{attribute 'linkalways'} 
{attribute 'no_explicit_call' := 'This FB is a CLASS and must be accessed using methods or properties'}
{attribute 'enable_dynamic_creation'}
FUNCTION_BLOCK _ETcVnSvmKernelType EXTENDS EnumDatatypeBase
VAR
	localData : ETcVnSvmKernelType;
	activeData : REFERENCE TO ETcVnSvmKernelType;
	enumBaseDatatype : _DINT(localData);
END_VAR

METHOD PRIVATE AddLocalEnumeration
VAR_INPUT
	Enumeration : T_MAXSTRING;
	Value : ETcVnSvmKernelType;
END_VAR
AddEnumeration(Enumeration, Value);
END_METHOD

PROPERTY PUBLIC Address : PVOID
GET
Address := ADR(activeData);
END_GET
END_PROPERTY

METHOD PUBLIC ClearReference
VAR_INPUT
END_VAR
activeData REF= localData;
SetBaseDatatypeReference();
END_METHOD

METHOD PUBLIC Clone : I_Datatype
VAR
    pClone : POINTER TO _ETcVnSvmKernelType;
END_VAR
pClone := __NEW(_ETcVnSvmKernelType(InitialValue := Value));
Clone := pClone^;
END_METHOD

METHOD FB_init : BOOL
VAR_INPUT
	bInitRetains : BOOL; // if TRUE, the retain variables are initialized (warm start / cold start)
	bInCopyCode : BOOL;  // if TRUE, the instance afterwards gets moved into the copy code (online change)
	InitialValue : ETcVnSvmKernelType;
END_VAR
localData := InitialValue;
AddBaseDatatype(enumBaseDatatype);
ClearReference();

AddLocalEnumeration('TCVN_SKT_LINEAR', ETcVnSvmKernelType.TCVN_SKT_LINEAR);
AddLocalEnumeration('TCVN_SKT_POLY', ETcVnSvmKernelType.TCVN_SKT_POLY);
AddLocalEnumeration('TCVN_SKT_RBF', ETcVnSvmKernelType.TCVN_SKT_RBF);
AddLocalEnumeration('TCVN_SKT_SIGMOID', ETcVnSvmKernelType.TCVN_SKT_SIGMOID);
AddLocalEnumeration('TCVN_SKT_CHI2', ETcVnSvmKernelType.TCVN_SKT_CHI2);
AddLocalEnumeration('TCVN_SKT_INTER', ETcVnSvmKernelType.TCVN_SKT_INTER);
END_METHOD

PROPERTY PUBLIC Identifier : T_MAXSTRING
GET
Identifier := 'ETcVnSvmKernelType';
END_GET
END_PROPERTY

METHOD IsEnumeratorValueEqual : BOOL
VAR_INPUT
	Enumerator : I_KeyValueForwardEnumerator;
END_VAR
VAR
	storedValue : ETcVnSvmKernelType;
END_VAR
IF NOT Enumerator.TryGet(storedValue) THEN
	RETURN;
END_IF

IsEnumeratorValueEqual := storedValue = activeData;
END_METHOD

METHOD PUBLIC MakeReferenceTo
VAR_INPUT
	ReferenceTarget : REFERENCE TO ETcVnSvmKernelType;
END_VAR
activeData REF= ReferenceTarget;
SetBaseDatatypeReference();
END_METHOD

METHOD PROTECTED SetBaseDatatypeReference
VAR_INPUT
END_VAR
enumBaseDatatype.MakeReferenceTo(activeData);
END_METHOD

PROPERTY PUBLIC Size : UDINT
GET
Size := SIZEOF(activeData);
END_GET
END_PROPERTY

METHOD TryMakeReferenceTo : BOOL
VAR_INPUT
	Target : I_Datatype;
END_VAR
VAR
	targetAsEnum : I_EnumDatatype;
	pTargetData : POINTER TO ETcVnSvmKernelType;
END_VAR
IF NOT Target.TryResolveAsEnumDatatype(targetAsEnum) THEN
	RETURN;
END_IF

IF targetAsEnum.Identifier <> Identifier THEN
	RETURN;
END_IF

pTargetData := Target.Address;
activeData REF= pTargetData^;
SetBaseDatatypeReference();
TryMakeReferenceTo := TRUE;
END_METHOD

PROPERTY PUBLIC Value : ETcVnSvmKernelType
GET
Value := activeData;
END_GET
SET
activeData := Value;
END_SET
END_PROPERTY

END_FUNCTION_BLOCK

(* stored: Version 1.1.0.1, ProductVersion 3.1.4024.13
   POU _ETcVnSvmKernelType: Id {d4918786-9cab-0cd6-2fcd-e628cd260273}, SpecialFunc None
   Folder Core: Id {512a4051-ce2d-08e0-3e05-45e6bff0025f}
   Folder Protected: Id {379efe20-a124-08ea-22a7-6ae65a05b89e}
   Folder Customize: Id {7ddb8890-7a2c-0ed9-32eb-8c3c1c2fa97c}
   Folder Constructor: Id {fcd5a4ca-c91d-0612-381f-e7e0e9d08047}
   Folder Private: Id {a9a80b6c-e641-03d0-2fa3-3e3ca7077f62}
   Folder Protected: Id {14f43d9a-4447-0614-0f11-bc60955d242b}
   Method AddLocalEnumeration: Id {b036fb34-c348-0c26-0e4c-9bda6ad7c67e}
   Property Address: Id {3cfcd777-4d74-0e79-1921-bcf5dc950f09}
   Get Get: Id {e96f154e-1a78-05de-23c4-a4aac86c2fc4}
   Method ClearReference: Id {2076ad69-a159-003c-045c-402f3267fda5}
   Method Clone: Id {62c5445e-85ae-0278-1045-f8b20dd75b01}
   Method FB_init: Id {363200be-d448-0413-224b-f9a2fa2c8541}
   Property Identifier: Id {7c1918a0-1ef6-05d7-146a-7ab05e9d0811}
   Get Get: Id {8d07742d-cd78-0be9-13ee-6c2f10d61f0c}
   Method IsEnumeratorValueEqual: Id {3e0367b2-34ba-06b7-3e5e-291ef48b21d8}
   Method MakeReferenceTo: Id {b1896ce3-d302-0310-2aec-ad9469df1070}
   Method SetBaseDatatypeReference: Id {e7b57660-8a96-0b5c-32c7-d6f0f74f2b6b}
   Property Size: Id {b05405a8-55d0-028f-3ba3-3c3d630b435e}
   Get Get: Id {759c2f2d-e774-0ab8-2a71-4d3239b7c561}
   Method TryMakeReferenceTo: Id {5537f957-8a00-05e1-2fa4-f921464ca333}
   Property Value: Id {9d332358-2bbb-0346-3533-f969f8cc28ce}
   Get Get: Id {bfb2b356-7527-03a3-002c-faef63a00b07}
   Set Set: Id {d44c2c32-608a-0a88-222b-8eea4c280e2b} *)
